PROGRAM MAIN
VAR
	nCounter : LREAL;
	rAmplitude : REAL;
	rPeriod	: REAL;
END_VAR

GVL.nCounter := GVL.nCounter + 0.02;

rAmplitude := 10*SIN(GVL.nCounter / 8);

rPeriod := 10*SIN(GVL.nCounter / 12);

GVL.sine := rAmplitude*SIN(GVL.nCounter / rPeriod);

END_PROGRAM

(* stored: Version 1.1.0.1, ProductVersion 3.1.4024.12
   POU MAIN: Id {fda9d826-ec2e-4388-ac70-0208ec875f25}, SpecialFunc None *)
